SUBAPPLICATION Uebung_020c2_sub (* DigitalInput_I1 auf DigitalOutput_Q1; E_TON Einschaltverzögert; Zeit eingeben und speichern. *)
  (* Standard: 61499-2; Description: Copyright (c) 2023 Meisterschulen am Ostbahnhof This program and the accompanying materials are made available under the terms of the Eclipse Public License 2.0 which is available at https://www.eclipse.org/legal/epl-2.0/ SPDX-License-Identifier: EPL-2.0 *)
  (* Version 1.0, 2023-10-31, Franz Höpfinger, Meisterschulen am Ostbahnhof *)
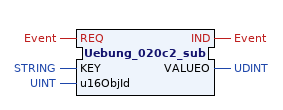
  EVENT_INPUT
    REQ;
  END_EVENT
  EVENT_OUTPUT
    IND;
  END_EVENT
  VAR_INPUT
    KEY : STRING;
    u16ObjId : UINT;
  END_VAR
  VAR_OUTPUT
    VALUEO : UDINT;
  END_VAR
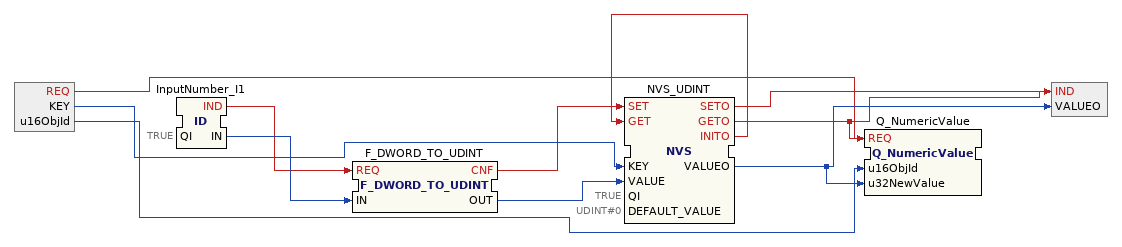
  FBS
    InputNumber_I1 : ID(QI := TRUE);
    F_DWORD_TO_UDINT : F_DWORD_TO_UDINT;
    NVS_UDINT : NVS(QI := TRUE, DEFAULT_VALUE := UDINT#0);
    Q_NumericValue : Q_NumericValue;
  END_FBS
  EVENT_CONNECTIONS
    InputNumber_I1.IND TO F_DWORD_TO_UDINT.REQ;
    REQ TO Q_NumericValue.REQ;
    F_DWORD_TO_UDINT.CNF TO NVS_UDINT.SET;
    NVS_UDINT.SETO TO IND;
    NVS_UDINT.GETO TO Q_NumericValue.REQ;
    NVS_UDINT.GETO TO IND;
    NVS_UDINT.INITO TO NVS_UDINT.GET;
  END_CONNECTIONS
  DATA_CONNECTIONS
    InputNumber_I1.IN TO F_DWORD_TO_UDINT.IN;
    u16ObjId TO Q_NumericValue.u16ObjId;
    KEY TO NVS_UDINT.KEY;
    F_DWORD_TO_UDINT.OUT TO NVS_UDINT.VALUE;
    NVS_UDINT.VALUEO TO Q_NumericValue.u32NewValue;
    NVS_UDINT.VALUEO TO VALUEO;
  END_CONNECTIONS
END_SUBAPPLICATION
